(* Logix 5000 project; controller RSL5k_18_Template_noLib Emulate 5570 rev 32.11; software revision 32.02; part 3 of 16 *)
(* tags used below, declared in another part *)
   PCmd_ClearCapt : BOOL;   // Program Command to Clear the captured min / max PV excursion values
   P_AIn : BOOL;   // Unique Parameter Name for auto - discovery
   Wrk_ValidONS : BOOL;   // Selected PV goes from Infinite or Not a Number to VALID
   OCmd_ResetAckAll : BOOL;   // Operator Command to Reset and Acknowledge all Alarms
   MCmd_InpPV : BOOL;   // Maintenance Command to use Input PV (normal)
   MCmd_SubstPV : BOOL;   // Maintenance Command to use Substitute PV (override input)
(* P_AIn, continued *)

ROUTINE Prescan   (* ladder *)
// Clear Ownership. clear "lurking" Commands
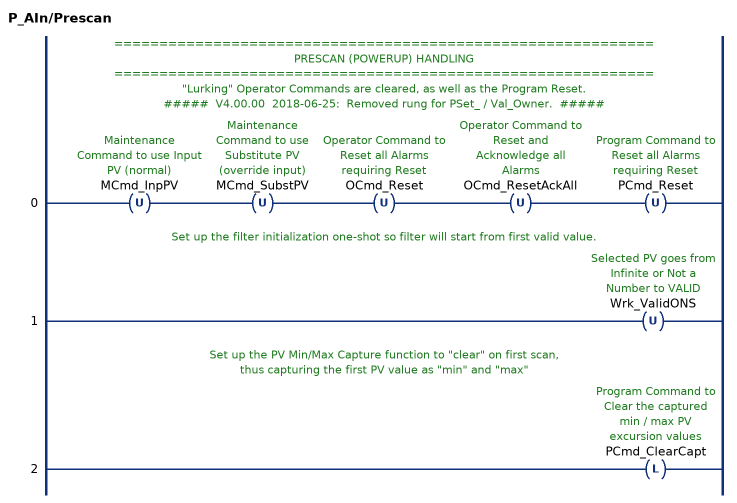
   // ============================================================
   // PRESCAN (POWERUP) HANDLING
   // ============================================================
   // "Lurking" Operator Commands are cleared, as well as the Program Reset.
   // #####  V4.00.00  2018-06-25:  Removed rung for PSet_ / Val_Owner.  #####
   0: OTU(MCmd_InpPV)OTU(MCmd_SubstPV)OTU(OCmd_Reset)OTU(OCmd_ResetAckAll)OTU(PCmd_Reset);
   // Set up the filter initialization one-shot so filter will start from first valid value.
   1: OTU(Wrk_ValidONS);
   // Set up the PV Min/Max Capture function to "clear" on first scan,
   // thus capturing the first PV value as "min" and "max"
   2: OTL(PCmd_ClearCapt);
END_ROUTINE
END_ADD_ON_INSTRUCTION

ADD_ON_INSTRUCTION P_Alarm   (* revision 4.10 .00 Release, vendor Rockwell Automation, ExecutePrescan, ExecuteEnableInFalse *)
// Alarm
// Revision note:
// See Instruction Help for a summary of changes, and see 4.10 Release Notes for details.
// Help:
// Copyright © Rockwell Automation, Inc.  All Rights Reserved.
// This instruction monitors one input condition and provides one Alarm with:
//   * configurable latching (reset required) and acknowledgement requirement
//   * configurable alarm severity
//       1 to 250       = Low  (blue, typ. informational)
//       251 to 500   = Medium  (yelllow, typ. warning)
//       501 to 750   = High  (red, typ. process exception)
//       751 to 1000 = Urgent  (magenta, typ. equip. fault)
//   * configurable minimum ON time (e.g., to ensure it is seen by the HMI)
//   * commands to suppress/unsuppress (Prog), shelve/unshelve (Oper)
//         and disable/enable (Maint) the alarm.
//   * configurable amount of time shelved to automatically unshelve an alarm
//   * FTA&E support for suppressed, shelved and disabled states (V7.0)
//   * a Maintenance "Test" command, which triggers the alarm for the minimum
//      alarm time for testing purposes.
// NOTE regarding parameter naming:
//   FTAE names (same as ALMD instruction) are used instead
//   of the ANSI/ISA 18.2-2009 names, as follows:
//    "Disabled" is the equivalent of "Out of Service" in ISA 18.2.
//       (The Disabled state is owned by Maintenance.)
//    "Suppressed" is the equivalent of "Suppressed by Design" in
//       ISA 18.2. (The Suppressed state is owned by Program logic.)
//    "Shelved" is the same as in ISA 18.2.
//       (The Shelved state is owned by Operator, but may be cleared
//       by Program logic based on time, shift change, etc.)
// This instruction is usually nested within other instructions, with one instance
// used for each Alarm generated by the containing instruction.  It may also be
// used as a standalone instruction for Alarm conditions generated by custom logic.
// FTAE Alarm Setup:
//   (object).(alarm).Com_AE.0:  Alarm to FTAE
//     .Com_AE.1:   Ack to/from FTAE
//     .Com_AE.3:   Shelved from FTAE Status
//     .Com_AE.4:   Shelve/Reshelve to FTAE Control (auto reset)
//     .Com_AE.5:   Unshelve to FTAE Control (auto reset)
//     .Com_AE.6:   Suppressed from FTAE Status
//     .Com_AE.7:   Suppress to FTAE Control (auto reset)
//     .Com_AE.8:   Unsuppress to FTAE Control (auto reset)
//     .Com_AE.9:   Disabled from FTAE Status
//     .Com_AE.10: Disable to FTAE Control (auto reset)
//     .Com_AE.11: Enable to FTAE Control (auto reset)
//    all other bits unused
//     .Cfg_MaxShelfT is also used in FTAE config.
//     .Cfg_Severity is used in FTAE for FTView 8.x and later.
// SUMMARY OF CHANGES FROM PREVIOUS VERSION (4.00.00)
// See 4.10 Release Notes for details.
// * Unmodified, up-rev only for Library 4.10.00
// SUMMARY OF CHANGES FROM PREVIOUS VERSION (3.5-07 Patch01)
// See 4.00 Release Notes for details.
// * Changed Inf_Lib and Inf_Type to HMI_Lib and HMI_Type.
// * Deleted Cfg_PCmdClear.  All Program Commands are now self-clearing.
// * Aligned ready bit naming with command bit names.
// * All OCmds/MCmds and ORdys/MRdys are now Local Tags.
// * Added Sts_RdyAck and Sts_RdyReset for use by containing objects.
// * Modified to remove Suppressed from the conditions which show the
//     "Inhibited" breadcrumb.
// * Added Inp_OoS for Out of Service from parent object's P_CmdSrc.
VAR_INPUT
   Inp : BOOL := 1; {visible}   // Alarm Condition Input 1=Alarm
   Inp_OoS : ALIAS FOR Com_AE.2;   // 1=Out of Service (from object's P_CmdSrc)
   Inp_Reset : BOOL; {visible}   // 1=Reset Alarm requiring reset
   Cfg_Exists : BOOL := 1;   // 1=Alarm configured to exist, 0=Does not exist, don't scan
   Cfg_ResetReqd : BOOL;   // 1=Latched Alarm, a Reset is required to clear this Alarm
   Cfg_AckReqd : BOOL := 1;   // 1=Acknowledge required for this Alarm
   Cfg_AllowShelve : BOOL := 1;   // 1=Allow Operator to Shelve this Alarm
   Cfg_AllowDisable : BOOL := 1;   // 1=Allow Maintenance to Disable this Alarm
   Cfg_Severity : DINT := 750;   // Alarm Severity: 1..250=Low, 251..500=Medium, 501..750=High, 751..1000=Urgent
   Cfg_MaxShelfT : DINT := 480;   // Auto unshelve after shelved this long (1..32767 minutes)
   Cfg_AlmMinOnT : DINT := 5;   // Minimum time Alm output stays on (sec)
   PCfg_AllowExist : BOOL := 1;   // 1=Alarm can be configured to exist, 0=other configs make alarm meaningless
   PCmd_Reset : BOOL;   // Program Command to Reset latched alarm
   PCmd_Ack : BOOL;   // Program Command to Acknowledge alarm
   PCmd_Suppress : BOOL;   // Program Command to Suppress by Design (inhibits new alarm)
   PCmd_Unsuppress : BOOL;   // Program Command to Unsuppress (allows new alarm)
   PCmd_Unshelve : BOOL;   // Program Command to Unshelve (e.g., on shift change)
END_VAR
VAR_OUTPUT
   Val_Notify : DINT; {access Read Only}   // Current Alarm Severity and Acknowledgement (enumeration)
   Val_SecToUnshelve : DINT; {access Read Only, visible}   // Number of Seconds until this alarm unshelves itself (mmm:ss)
   Val_MinToUnshelve : DINT; {access Read Only, visible}   // Number of minutes until this alarm unshelves itself (mmm:ss)
   Alm : ALIAS FOR Com_AE.0; {visible}   // Alarm output 1=In Alarm
   Ack : ALIAS FOR Com_AE.1; {visible}   // Alarm acknowledged status: 1=Ack rcvd
   Shelved : ALIAS FOR Com_AE.3; {visible}   // 1=Alarm has been Shelved by Operator (inhibits new alarm)
   Suppressed : ALIAS FOR Com_AE.6; {visible}   // 1=Alarm has been Suppressed by Program (inhibits new alarm)
   Disabled : ALIAS FOR Com_AE.9; {visible}   // 1=Alarm has been Disabled by Maintanance (inhibits new alarm)
   Sts_AlmInh : BOOL; {access Read Only}   // 1=Alarm has been suppressed, shelved or disabled, display "I" icon
   Sts_RdyReset : ALIAS FOR ORdy_Reset; {access Read Only}   // 1=A latched alarm or shed condition is ready to be reset
   Sts_RdyAck : ALIAS FOR ORdy_Ack; {access Read Only}   // 1=An alarm is ready to be acknowledged
   Sts_Err : BOOL; {access Read Only}   // 1=Error in Config: see detail Err_ bits for reason
   Err_Timer : BOOL; {access Read Only}   // 1=Error in Config: Alarm Min On Time, Shelf Time (use 0 to 2147483)
   Err_Severity : BOOL; {access Read Only}   // 1=Error in Config: Invalid Severity (use 1 to 4)
   P_Alarm : BOOL;   // Unique Parameter Name for auto - discovery
END_VAR
VAR
   Wrk_Alm : BOOL; {access None}   // Internal Alarm Status
   Wrk_Suppressed : BOOL; {access None}   // Internal Alarm Suppressed Status
   Wrk_AlmMinOnT : TIMER := (PRE := 5000); {access None}   // Alarm output minimum ON time to be seen by alarm server
   Wrk_AutoAckT : TIMER := (PRE := 5000); {access None}   // Time to clear Ack bit when Ack not required
   Wrk_ShelfT : TIMER; {access Read Only}   // Time to auto Unshelve a Shelved Alarm
   HMI_Tab : SINT;   // Tab to display (FTView ME)
   Com_AE : INT := 2#0000_0000_0000_0010;   // Communication with HMI / Alarm/Event Server (see bit descriptions)
        .0   // Alarm to AE
        .10   // Disable to AE Control
        .11   // Enable to AE Control
        .12   // (not used)
        .13   // (not used)
        .14   // (not used)
        .15   // (not used)
        .1   // Acked from AE Status, Ack to AE Control
        .2   // Out of Service (from parent object's P_CmdSrc)
        .3   // Shelved from AE Status
        .4   // Shelve to AE Control
        .5   // Unshelve to AE Control
        .6   // Suppressed from AE Status
        .7   // Suppress to AE Control
        .8   // Unsuppress to AE Control
        .9   // Disabled from AE Status
   Cfg_Tag : STRING_20 := 'P_Alarm';   // Alarm Tag Text (e.g., "LAHH-101")
   Cfg_Cond : STRING_20 := 'Alarm Condition';   // Alarm Condition Text (e.g., "High-High PV")
   Wrk_SecToUnshelve : DINT; {access None}   // Number of seconds until this alarm unshelves itself
   HMI_Lib : STRING_12 := 'RA-BAS'; {access Read Only}   // Display Library for Faceplate call-up
   HMI_Type : STRING_16 := 'P_Alarm'; {access Read Only}   // Must contain AOI name, used for HMI and Information S/W
   ORdy_Unshelve : BOOL; {access Read Only}   // 1=Ready for OCmd_Unshelve (enables HMI button)
   ORdy_Shelve : BOOL; {access Read Only}   // 1=Ready for OCmd_Shelve (enables HMI button)
   MRdy_Test : BOOL; {access Read Only}   // 1=Ready for MCmd_Test (enables HMI button)
   MRdy_Enable : BOOL; {access Read Only}   // 1=Ready for MCmd_Enable (enables HMI button)
   MRdy_Disable : BOOL; {access Read Only}   // 1=Ready for MCmd_Disable (enables HMI button)
   OCmd_Unshelve : BOOL;   // Operator Command to Unshelve alarm (allows new alarm)
   OCmd_Shelve : BOOL;   // Operator Command to Shelve Alarm (inhibits new alarm)
   OCmd_Ack : BOOL;   // Operator Command to Acknowledge alarm
   OCmd_Reset : BOOL;   // Operator Command to Reset latched alarm
   MCmd_Test : BOOL;   // Maintenance Command to Test alarm (issued for minimum alarm time)
   MCmd_Enable : BOOL;   // Maintenance Command to Enable alarm (allows new alarm)
   MCmd_Disable : BOOL;   // Maintenance Command to Disable alarm (inhibits new alarm)
   ORdy_Ack : BOOL; {access Read Only}   // 1=Ready for OCmd_Ack (enables HMI button)
   ORdy_Reset : BOOL; {access Read Only}   // 1=Ready for OCmd_Reset (enables HMI button)
END_VAR

ROUTINE EnableInFalse   (* ladder *)
// Perform Alarm processing, but Invert Alarm Input ("Inp") for use on LD rung (EnableIn False)
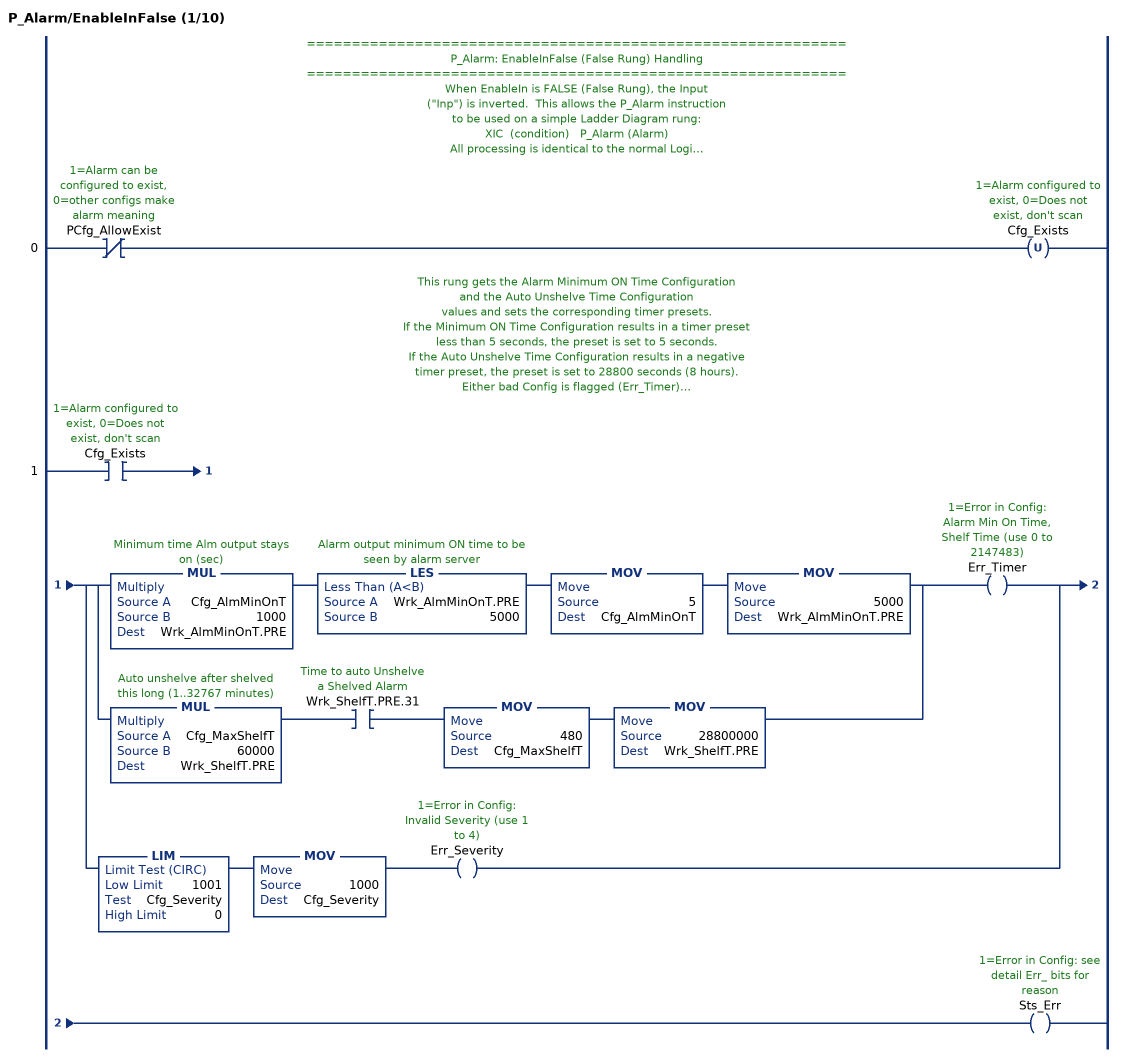
   // ============================================================
   // P_Alarm: EnableInFalse (False Rung) Handling
   // ============================================================
   // When EnableIn is FALSE (False Rung), the Input
   // ("Inp") is inverted.  This allows the P_Alarm instruction
   // to be used on a simple Ladder Diagram rung:
   // XIC  (condition)   P_Alarm (Alarm)
   // All processing is identical to the normal Logic
   // routine, except references to Inp are inverted!
   // ============================================================
   // CONFIGURATION
   // ============================================================
   // In the object containing this alarm, other configuration (such as not having
   // any limit switches) may make this particular alarm meaningless.
   // The Program Configuration "Allow Exist" is used to hide this alarm
   // on the object's faceplate and other graphics, and forces the Cfg_Exist to 0.
   0: XIO(PCfg_AllowExist)OTU(Cfg_Exists);
   // This rung gets the Alarm Minimum ON Time Configuration
   // and the Auto Unshelve Time Configuration
   // values and sets the corresponding timer presets.
   // If the Minimum ON Time Configuration results in a timer preset
   // less than 5 seconds, the preset is set to 5 seconds.
   // If the Auto Unshelve Time Configuration results in a negative
   // timer preset, the preset is set to 28800 seconds (8 hours).
   // Either bad Config is flagged (Err_Timer).
   // Bad Config is also flagged if the Cfg_Severity is out of range (valid = 1..1000) (Err_Severity).
   1: XIC(Cfg_Exists)[[MUL(Cfg_AlmMinOnT,1000,Wrk_AlmMinOnT.PRE) LES(Wrk_AlmMinOnT.PRE,5000) MOV(5,Cfg_AlmMinOnT) MOV(5000,Wrk_AlmMinOnT.PRE) ,MUL(Cfg_MaxShelfT,60000,Wrk_ShelfT.PRE) XIC(Wrk_ShelfT.PRE.31) MOV(480,Cfg_MaxShelfT) MOV(28800000,Wrk_ShelfT.PRE) ] OTE(Err_Timer) ,LIM(1001,Cfg_Severity,0) MOV(1000,Cfg_Severity) OTE(Err_Severity) ]OTE(Sts_Err);
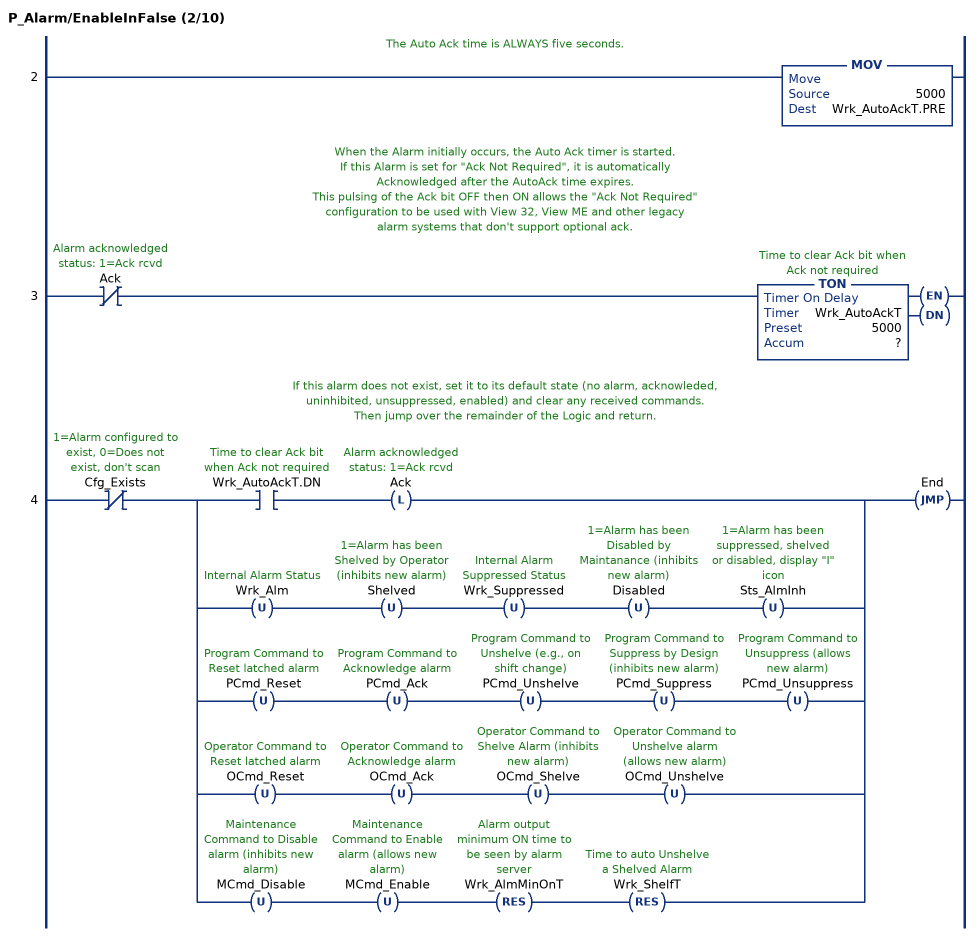
   // The Auto Ack time is ALWAYS five seconds.
   2: MOV(5000,Wrk_AutoAckT.PRE);
   // When the Alarm initially occurs, the Auto Ack timer is started.
   // If this Alarm is set for "Ack Not Required", it is automatically
   // Acknowledged after the AutoAck time expires.
   // This pulsing of the Ack bit OFF then ON allows the "Ack Not Required"
   // configuration to be used with View 32, View ME and other legacy
   // alarm systems that don't support optional ack.
   3: XIO(Ack)TON(Wrk_AutoAckT,?,?);
   // If this alarm does not exist, set it to its default state (no alarm, acknowleded,
   // uninhibited, unsuppressed, enabled) and clear any received commands.
   // Then jump over the remainder of the Logic and return.
   4: XIO(Cfg_Exists)[XIC(Wrk_AutoAckT.DN) OTL(Ack) ,OTU(Wrk_Alm) OTU(Shelved) OTU(Wrk_Suppressed) OTU(Disabled) OTU(Sts_AlmInh) ,OTU(PCmd_Reset) OTU(PCmd_Ack) OTU(PCmd_Unshelve) OTU(PCmd_Suppress) OTU(PCmd_Unsuppress) ,OTU(OCmd_Reset) OTU(OCmd_Ack) OTU(OCmd_Shelve) OTU(OCmd_Unshelve) ,OTU(MCmd_Disable) OTU(MCmd_Enable) RES(Wrk_AlmMinOnT) RES(Wrk_ShelfT) ]JMP(End);
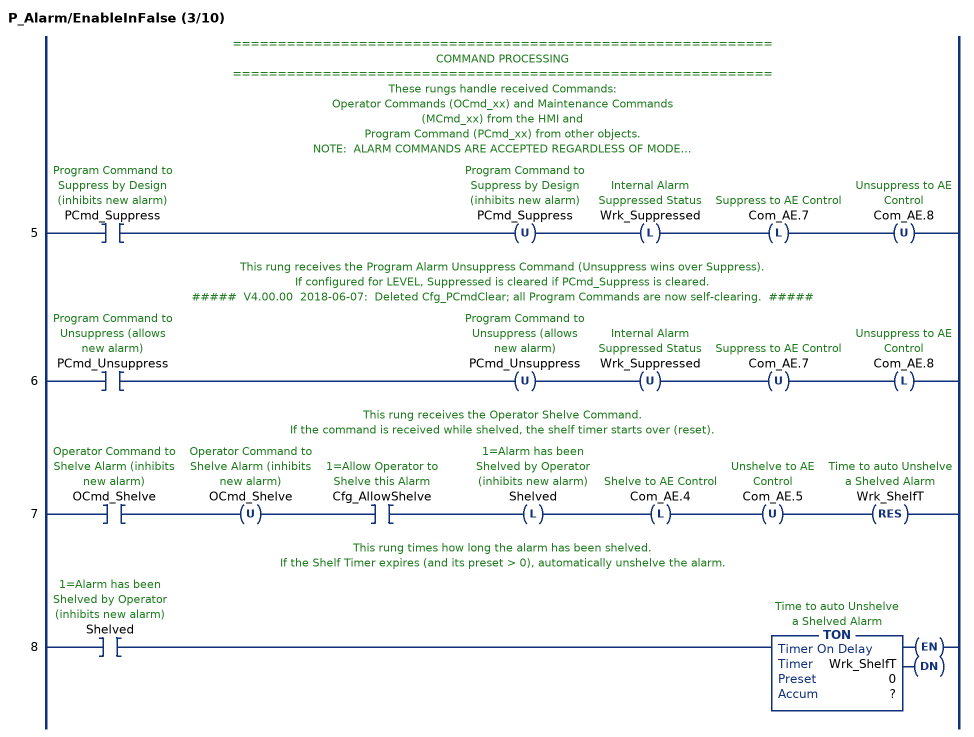
   // ============================================================
   // COMMAND PROCESSING
   // ============================================================
   // These rungs handle received Commands:
   // Operator Commands (OCmd_xx) and Maintenance Commands
   // (MCmd_xx) from the HMI and
   // Program Command (PCmd_xx) from other objects.
   // NOTE:  ALARM COMMANDS ARE ACCEPTED REGARDLESS OF MODE.
   // This rung receives the Program Alarm Inhibit Command.
   // If configured for EDGE, the Command is cleared.
   // #####  V4.00.00  2018-06-07:  Deleted Cfg_PCmdClear; all Program Commands are now self-clearing.  #####
   5: XIC(PCmd_Suppress)OTU(PCmd_Suppress)OTL(Wrk_Suppressed)OTL(Com_AE.7)OTU(Com_AE.8);
   // This rung receives the Program Alarm Unsuppress Command (Unsuppress wins over Suppress).
   // If configured for LEVEL, Suppressed is cleared if PCmd_Suppress is cleared.
   // #####  V4.00.00  2018-06-07:  Deleted Cfg_PCmdClear; all Program Commands are now self-clearing.  #####
   6: XIC(PCmd_Unsuppress)OTU(PCmd_Unsuppress)OTU(Wrk_Suppressed)OTU(Com_AE.7)OTL(Com_AE.8);
   // This rung receives the Operator Shelve Command.
   // If the command is received while shelved, the shelf timer starts over (reset).
   7: XIC(OCmd_Shelve)OTU(OCmd_Shelve)XIC(Cfg_AllowShelve)OTL(Shelved)OTL(Com_AE.4)OTU(Com_AE.5)RES(Wrk_ShelfT);
   // This rung times how long the alarm has been shelved.
   // If the Shelf Timer expires (and its preset > 0), automatically unshelve the alarm.
   8: XIC(Shelved)TON(Wrk_ShelfT,?,?);
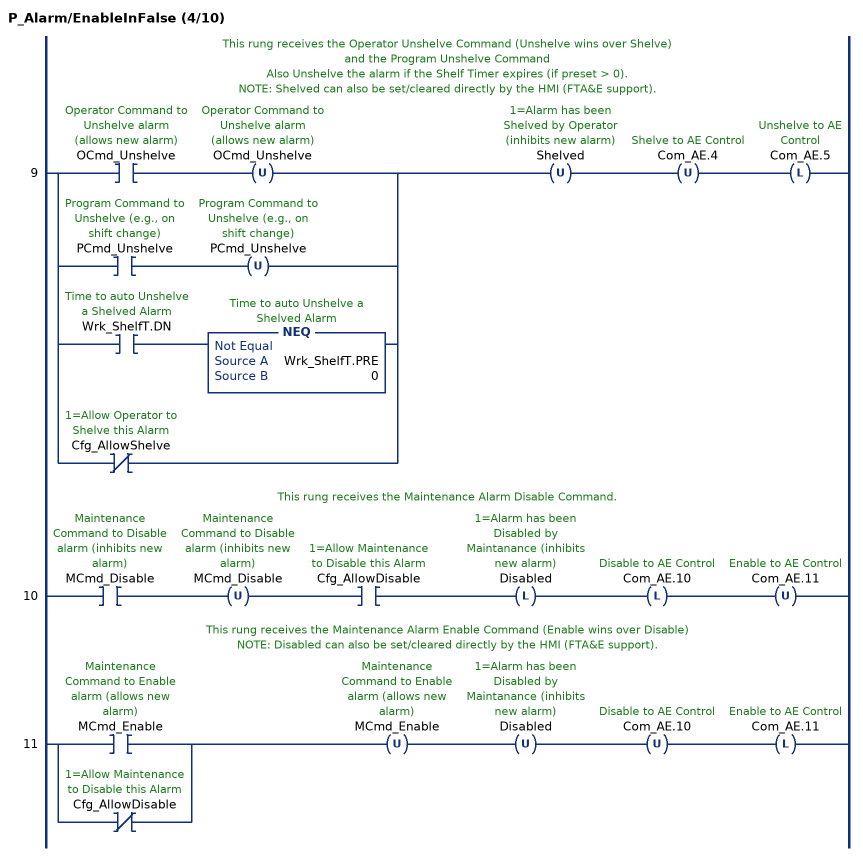
   // This rung receives the Operator Unshelve Command (Unshelve wins over Shelve)
   // and the Program Unshelve Command
   // Also Unshelve the alarm if the Shelf Timer expires (if preset > 0).
   // NOTE: Shelved can also be set/cleared directly by the HMI (FTA&E support).
   9: [XIC(OCmd_Unshelve) OTU(OCmd_Unshelve) ,XIC(PCmd_Unshelve) OTU(PCmd_Unshelve) ,XIC(Wrk_ShelfT.DN) NEQ(Wrk_ShelfT.PRE,0) ,XIO(Cfg_AllowShelve) ]OTU(Shelved)OTU(Com_AE.4)OTL(Com_AE.5);
   // This rung receives the Maintenance Alarm Disable Command.
   10: XIC(MCmd_Disable)OTU(MCmd_Disable)XIC(Cfg_AllowDisable)OTL(Disabled)OTL(Com_AE.10)OTU(Com_AE.11);
   // This rung receives the Maintenance Alarm Enable Command (Enable wins over Disable)
   // NOTE: Disabled can also be set/cleared directly by the HMI (FTA&E support).
   11: [XIC(MCmd_Enable) ,XIO(Cfg_AllowDisable) ]OTU(MCmd_Enable)OTU(Disabled)OTU(Com_AE.10)OTL(Com_AE.11);
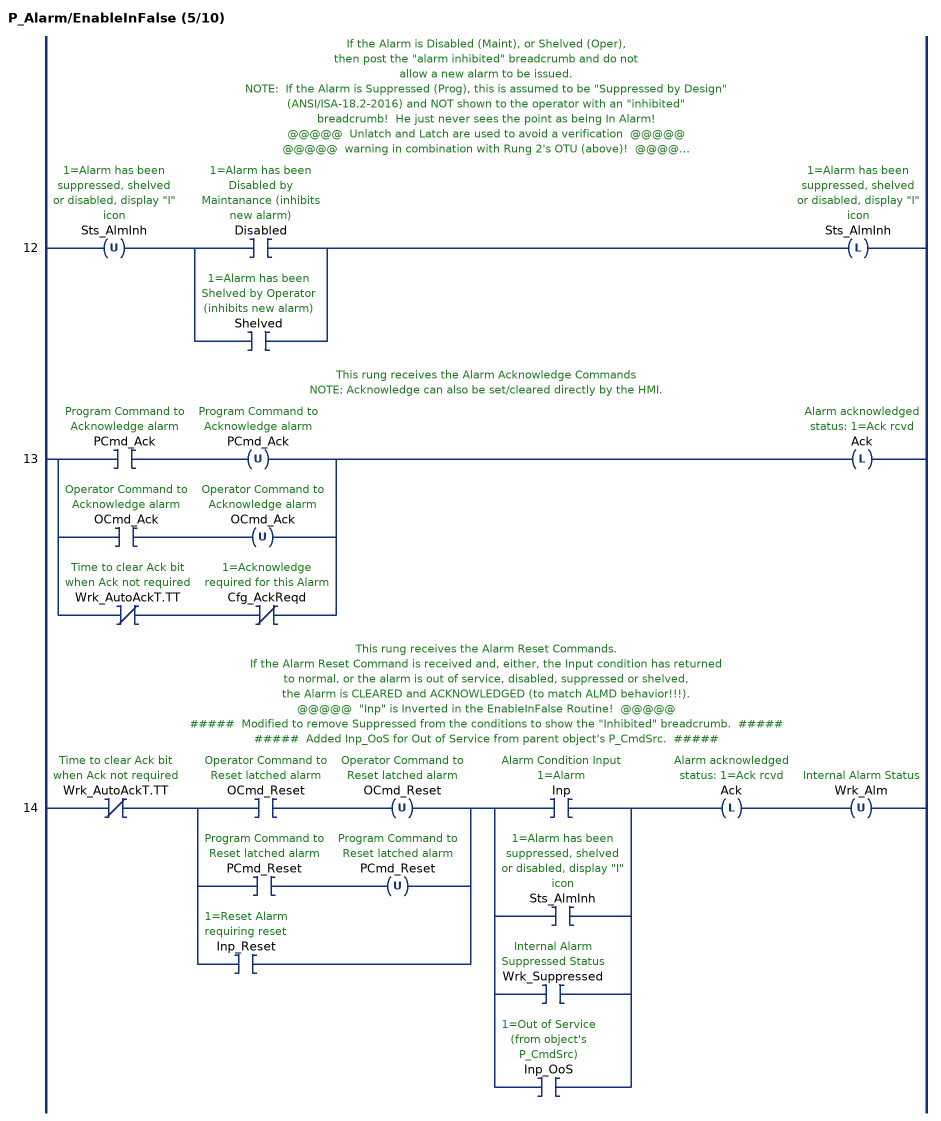
   // If the Alarm is Disabled (Maint), or Shelved (Oper),
   // then post the "alarm inhibited" breadcrumb and do not
   // allow a new alarm to be issued.
   // NOTE:  If the Alarm is Suppressed (Prog), this is assumed to be "Suppressed by Design"
   // (ANSI/ISA-18.2-2016) and NOT shown to the operator with an "inhibited"
   // breadcrumb!  He just never sees the point as being In Alarm!
   // @@@@@  Unlatch and Latch are used to avoid a verification  @@@@@
   // @@@@@  warning in combination with Rung 2's OTU (above)!  @@@@@
   // #####  V4.00.00  2018-06-07:  Modified to remove Suppressed from the conditions to show the "Inhibited" breadcrumb.  #####
   12: OTU(Sts_AlmInh)[XIC(Disabled) ,XIC(Shelved) ]OTL(Sts_AlmInh);
   // This rung receives the Alarm Acknowledge Commands
   // NOTE: Acknowledge can also be set/cleared directly by the HMI.
   13: [XIC(PCmd_Ack) OTU(PCmd_Ack) ,XIC(OCmd_Ack) OTU(OCmd_Ack) ,XIO(Wrk_AutoAckT.TT) XIO(Cfg_AckReqd) ]OTL(Ack);
   // This rung receives the Alarm Reset Commands.
   // If the Alarm Reset Command is received and, either, the Input condition has returned
   // to normal, or the alarm is out of service, disabled, suppressed or shelved,
   // the Alarm is CLEARED and ACKNOWLEDGED (to match ALMD behavior!!!).
   // @@@@@  "Inp" is Inverted in the EnableInFalse Routine!  @@@@@
   // #####  Modified to remove Suppressed from the conditions to show the "Inhibited" breadcrumb.  #####
   // #####  Added Inp_OoS for Out of Service from parent object's P_CmdSrc.  #####
   14: XIO(Wrk_AutoAckT.TT)[XIC(OCmd_Reset) OTU(OCmd_Reset) ,XIC(PCmd_Reset) OTU(PCmd_Reset) ,XIC(Inp_Reset) ][XIC(Inp) ,XIC(Sts_AlmInh) ,XIC(Wrk_Suppressed) ,XIC(Inp_OoS) ]OTL(Ack)OTU(Wrk_Alm);
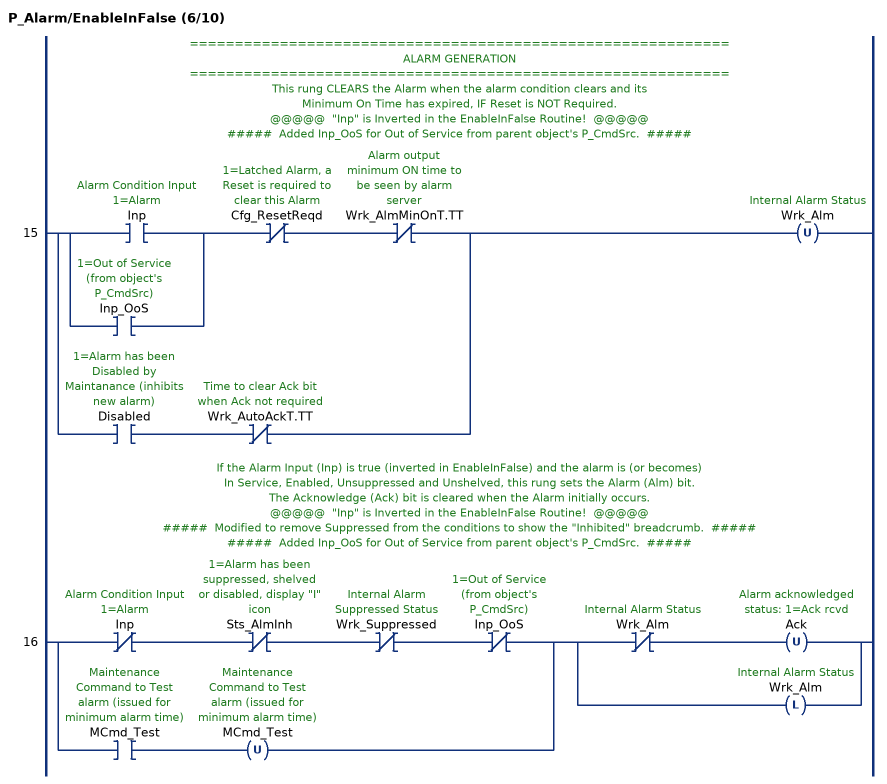
   // ============================================================
   // ALARM GENERATION
   // ============================================================
   // This rung CLEARS the Alarm when the alarm condition clears and its
   // Minimum On Time has expired, IF Reset is NOT Required.
   // @@@@@  "Inp" is Inverted in the EnableInFalse Routine!  @@@@@
   // #####  Added Inp_OoS for Out of Service from parent object's P_CmdSrc.  #####
   15: [[XIC(Inp) ,XIC(Inp_OoS) ] XIO(Cfg_ResetReqd) XIO(Wrk_AlmMinOnT.TT) ,XIC(Disabled) XIO(Wrk_AutoAckT.TT) ]OTU(Wrk_Alm);
   // If the Alarm Input (Inp) is true (inverted in EnableInFalse) and the alarm is (or becomes)
   // In Service, Enabled, Unsuppressed and Unshelved, this rung sets the Alarm (Alm) bit.
   // The Acknowledge (Ack) bit is cleared when the Alarm initially occurs.
   // @@@@@  "Inp" is Inverted in the EnableInFalse Routine!  @@@@@
   // #####  Modified to remove Suppressed from the conditions to show the "Inhibited" breadcrumb.  #####
   // #####  Added Inp_OoS for Out of Service from parent object's P_CmdSrc.  #####
   16: [XIO(Inp) XIO(Sts_AlmInh) XIO(Wrk_Suppressed) XIO(Inp_OoS) ,XIC(MCmd_Test) OTU(MCmd_Test) ][XIO(Wrk_Alm) OTU(Ack) ,OTL(Wrk_Alm) ];
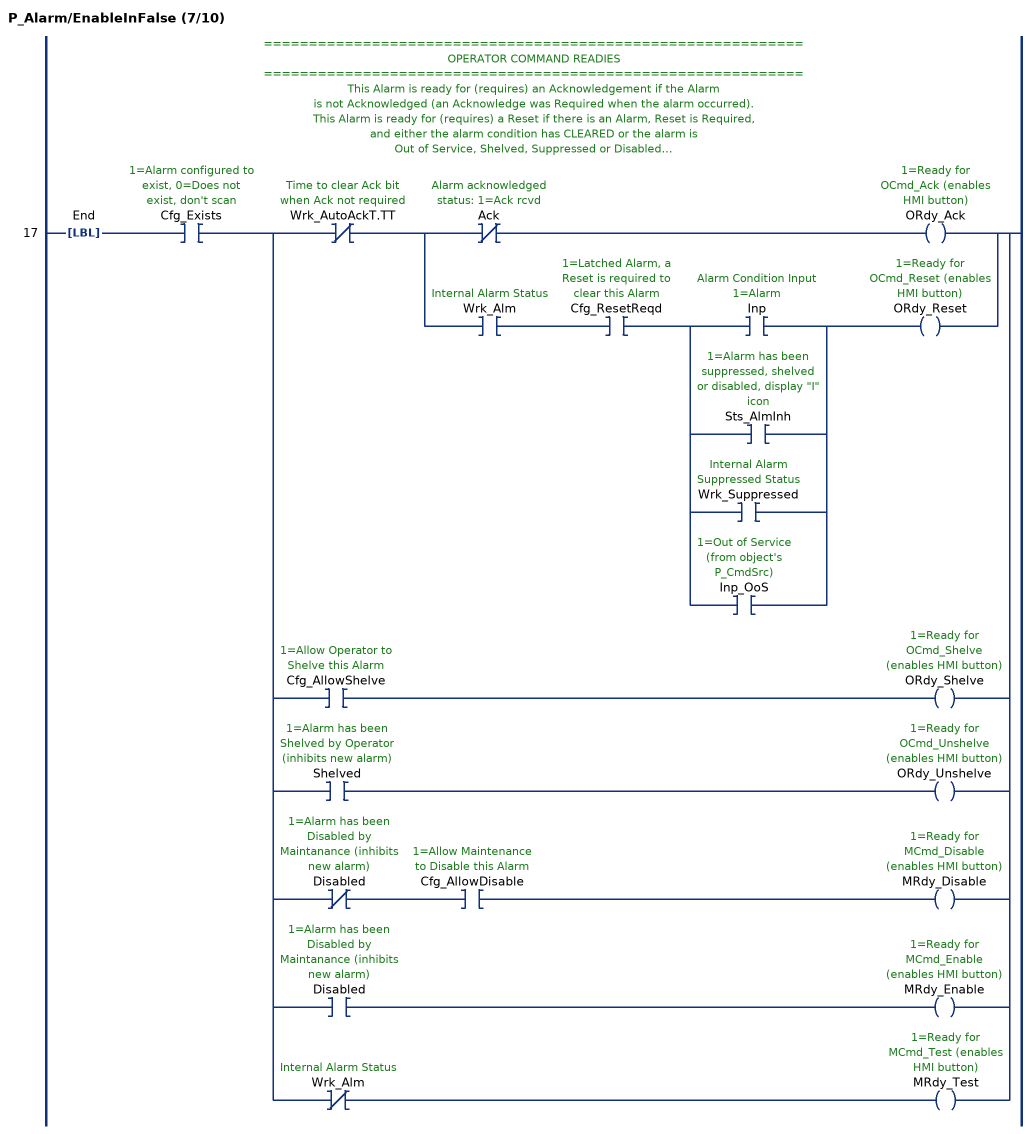
   // ============================================================
   // OPERATOR COMMAND READIES
   // ============================================================
   // This Alarm is ready for (requires) an Acknowledgement if the Alarm
   // is not Acknowledged (an Acknowledge was Required when the alarm occurred).
   // This Alarm is ready for (requires) a Reset if there is an Alarm, Reset is Required,
   // and either the alarm condition has CLEARED or the alarm is
   // Out of Service, Shelved, Suppressed or Disabled.
   // .
   // If the Alarm is NOT Shelved, it is ready for Shelve.
   // If the Alarm IS Shelved, it is ready for Unshelve.
   // If the Alarm is NOT Disabled, it is ready for Disable.
   // If the Alarm IS Disabled, it is ready for Enable.
   // NOTE: This rung appears before the Values/Status rung because the Rdy_Reset
   // condition is used to eliminate redundant logic in the rung below for Val_Notify.0.
   // @@@@@  "Inp" is Inverted in the EnableInFalse Routine!  @@@@@
   // #####  V4.00.00  2018-06-07:  Aligned ready bit naming with command bit names.  #####
   // #####  All OCmds/MCmds and ORdys/MRdys are now Local Tags.  #####
   // #####  Added Sts_RdyAck and Sts_ResetReqd for use by containing objects.  #####
   // #####  Modified to remove Suppressed from the conditions to show the "Inhibited" breadcrumb.  #####
   // #####  Added Inp_OoS for Out of Service from parent object's P_CmdSrc.  #####
   17: LBL(End)XIC(Cfg_Exists)[XIO(Wrk_AutoAckT.TT) [XIO(Ack) OTE(ORdy_Ack) ,XIC(Wrk_Alm) XIC(Cfg_ResetReqd) [XIC(Inp) ,XIC(Sts_AlmInh) ,XIC(Wrk_Suppressed) ,XIC(Inp_OoS) ] OTE(ORdy_Reset) ] ,XIC(Cfg_AllowShelve) OTE(ORdy_Shelve) ,XIC(Shelved) OTE(ORdy_Unshelve) ,XIO(Disabled) XIC(Cfg_AllowDisable) OTE(MRdy_Disable) ,XIC(Disabled) OTE(MRdy_Enable) ,XIO(Wrk_Alm) OTE(MRdy_Test) ];
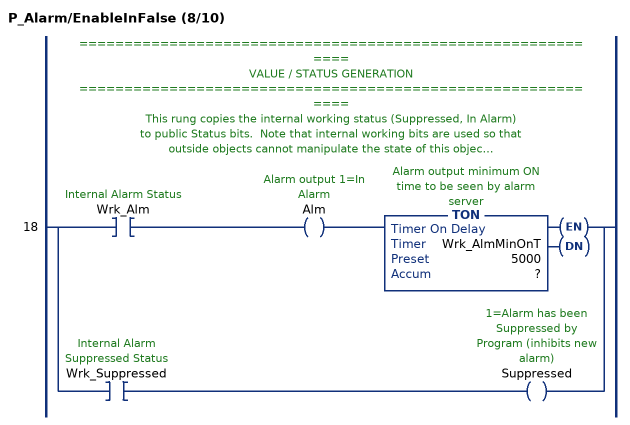
   // ============================================================
   // VALUE / STATUS GENERATION
   // ============================================================
   // This rung copies the internal working status (Suppressed, In Alarm)
   // to public Status bits.  Note that internal working bits are used so that
   // outside objects cannot manipulate the state of this object
   // by setting/clearing its Status and Alarm bits.
   // Public Status is generated for:
   // Alarm (with minimum ON time to be seen by polling)
   // Alarm Suppressed
   // Unsuppressed, Unshelved and Enabled are generated for HMI (FTVSE 7).
   // (Ack, Shelved and Disabled can be set/cleared by the HMI directly.
   // Note that these bits are "read/write" outputs in the parameter definition.)
   18: [XIC(Wrk_Alm) OTE(Alm) TON(Wrk_AlmMinOnT,?,?) ,XIC(Wrk_Suppressed) OTE(Suppressed) ];
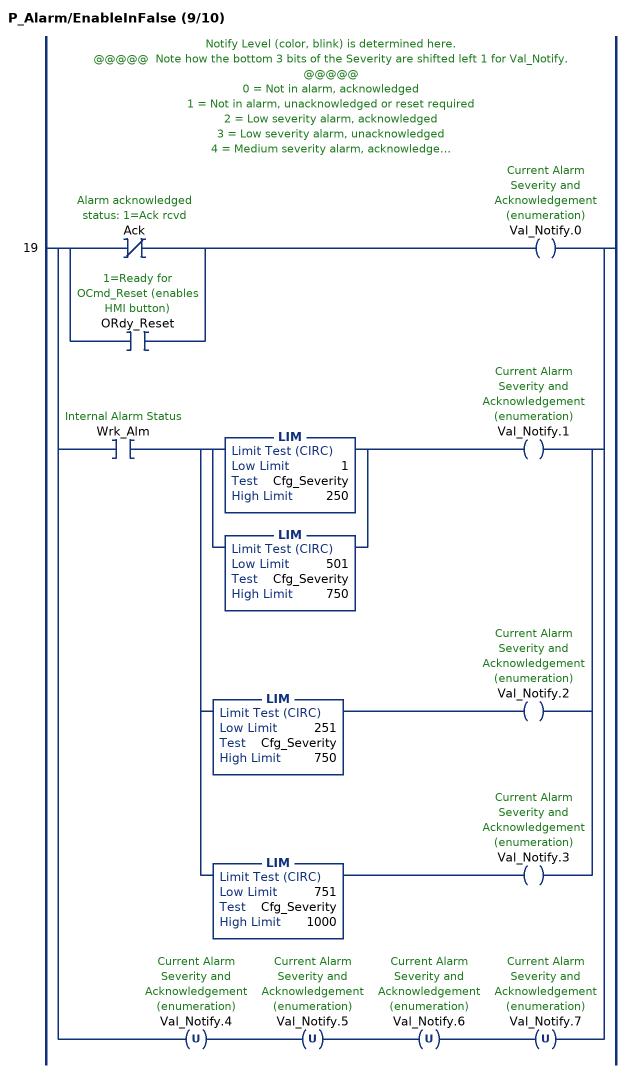
   // Notify Level (color, blink) is determined here.
   // @@@@@  Note how the bottom 3 bits of the Severity are shifted left 1 for Val_Notify.  @@@@@
   // 0 = Not in alarm, acknowledged
   // 1 = Not in alarm, unacknowledged or reset required
   // 2 = Low severity alarm, acknowledged
   // 3 = Low severity alarm, unacknowledged
   // 4 = Medium severity alarm, acknowledged
   // 5 = Medium severity alarm, unacknowledged
   // 6 = High severity alarm, acknowledged
   // 7 = High severity alarm, unacknowledged
   // 8 = Urgent severity alarm, acknowledged
   // 9 = Urgent severity alarm, unacknowledged
   // NOTE that the alarm bell icon will blink, even though the alarm is Acknowledged,
   // if an Alarm Reset is required (to get the Operator's attention).
   19: [[XIO(Ack) ,XIC(ORdy_Reset) ] OTE(Val_Notify.0) ,XIC(Wrk_Alm) [[LIM(1,Cfg_Severity,250) ,LIM(501,Cfg_Severity,750) ] OTE(Val_Notify.1) ,LIM(251,Cfg_Severity,750) OTE(Val_Notify.2) ,LIM(751,Cfg_Severity,1000) OTE(Val_Notify.3) ] ,OTU(Val_Notify.4) OTU(Val_Notify.5) OTU(Val_Notify.6) OTU(Val_Notify.7) ];
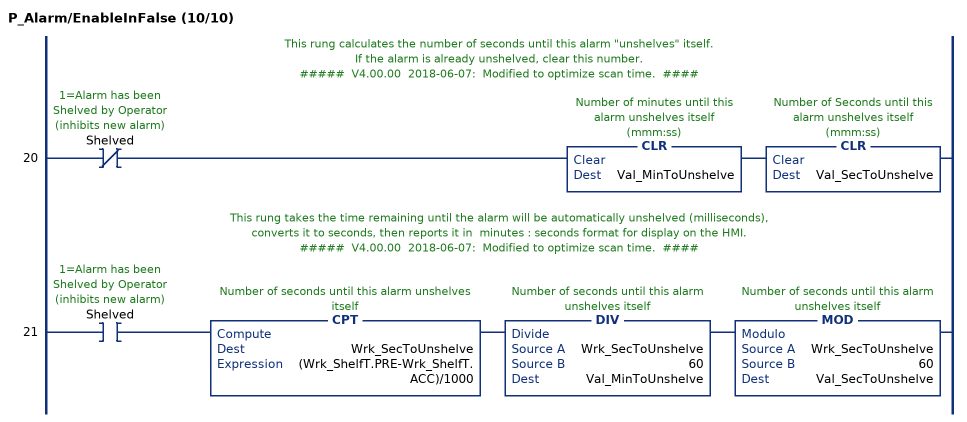
   // This rung calculates the number of seconds until this alarm "unshelves" itself.
   // If the alarm is already unshelved, clear this number.
   // #####  V4.00.00  2018-06-07:  Modified to optimize scan time.  ####
   20: XIO(Shelved)CLR(Val_MinToUnshelve)CLR(Val_SecToUnshelve);
   // This rung takes the time remaining until the alarm will be automatically unshelved (milliseconds),
   // converts it to seconds, then reports it in  minutes : seconds format for display on the HMI.
   // #####  V4.00.00  2018-06-07:  Modified to optimize scan time.  ####
   21: XIC(Shelved)CPT(Wrk_SecToUnshelve,(Wrk_ShelfT.PRE-Wrk_ShelfT.ACC)/1000)DIV(Wrk_SecToUnshelve,60,Val_MinToUnshelve)MOD(Wrk_SecToUnshelve,60,Val_SecToUnshelve);
END_ROUTINE

ROUTINE Logic   (* ladder *)
// Perform Alarm processing: delay, latch/reset, acknowledge, enable/disable, inhibit/uninhibit, suppress/unsuppress
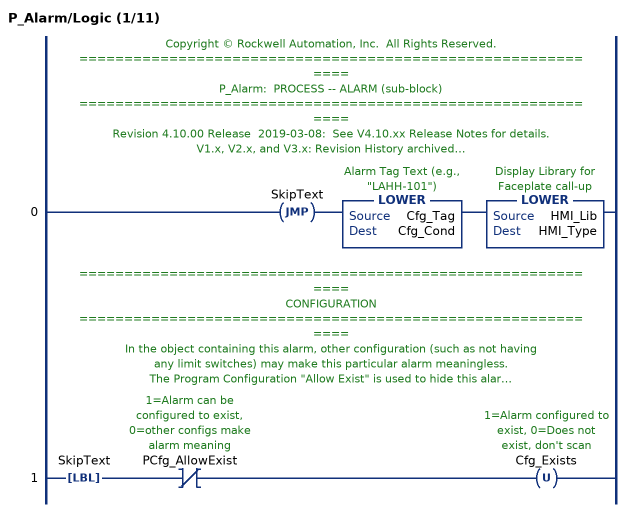
   // Copyright © Rockwell Automation, Inc.  All Rights Reserved.
   // ============================================================
   // P_Alarm:  PROCESS -- ALARM (sub-block)
   // ============================================================
   // Revision 4.10.00 Release  2019-03-08:  See V4.10.xx Release Notes for details.
   // V1.x, V2.x, and V3.x: Revision History archived.
   // V4.00.00  2018-06-07:  Changed Inf_ items to HMI_. Deleted Cfg_PCmdClear.
   // Aligned ready bit naming with command bit names.
   // All OCmds/MCmds and ORdys/MRdys are now Local Tags.
   // Added Sts_RdyAck and Sts_RdyReset for use by containing objects.
   // Modified to remove Suppressed from the conditions which show
   // the "Inhibited" breadcrumb.
   // Added Inp_OoS for Out of Service from parent object's P_CmdSrc.
   // V4.10.00  2019-03-08:  Unmodified, up-rev only for Library 4.10.00
   // ============================================================
   // This instruction monitors one input condition and provides one Alarm with:
   //   * configurable latching (reset required) and acknowledgement requirement
   //   * configurable alarm severity
   // 1..250 = Low  (blue, typ. informational)
   // 251-500 = Medium  (yelllow, typ. warning)
   // 501-750 = High  (red, typ. process exception)
   // 751-1000 = Urgent  (magenta, typ. equip. fault)
   // * configurable minimum ON time (e.g., to ensure it is seen by the HMI)
   // * commands to suppress/unsuppress (Prog), shelve/unshelve (Oper)
   // and disable/enable (Maint) the alarm.
   // * configurable amount of time shelved to automatically unshelve an alarm
   // * FTA&E support for suppressed, shelved and disabled states (V7.0)
   // NOTE regarding parameter naming:
   // FTA&E names (same as ALMD instruction) are used instead
   // of the ANSI/ISA 18.2-2016 names, as follows:
   // "Disabled" is the equivalent of "Out of Service" in ISA 18.2.
   // (the Disabled state is owned by Maintenance)
   // "Suppressed" is the equivalent of "Suppressed by Design" in ISA 18.2.
   // (the Suppressed state is owned by Program logic)
   // "Shelved" is the same as in ISA 18.2.
   // (the Shelved state is owned by Operator, but may be cleared
   // by Program logic based on time, shift change, etc.)
   // This instruction is usually nested within other instructions, with one instance
   // used for each Alarm generated by the containing instruction.  It may also be
   // used as a standalone instruction for Alarm conditions generated by custom logic.
   // ________________________________________
   // FTAE Alarm Setup:
   // ________________________________________
   // (object).(alarm).Com_AE.0:  Alarm to FTAE
   // .Com_AE.1:   Ack to/from FTAE
   // .Com_AE.2:  Out of Service (from object's P_CmdSrc)
   // .Com_AE.3:   Shelved from FTAE Status
   // .Com_AE.4:   Shelve/Reshelve to FTAE Control (auto reset)
   // .Com_AE.5:   Unshelve to FTAE Control (auto reset)
   // .Com_AE.6:   Suppressed from FTAE Status
   // .Com_AE.7:   Suppress to FTAE Control (auto reset)
   // .Com_AE.8:   Unsuppress to FTAE Control (auto reset)
   // .Com_AE.9:   Disabled from FTAE Status
   // .Com_AE.10: Disable to FTAE Control (auto reset)
   // .Com_AE.11: Enable to FTAE Control (auto reset)
   // all other bits unused
   //     .Cfg_MaxShelfT is also used in FTAE config.
   // .Cfg_Severity is used by FTAE in FTView 8.x.
   // ============================================================
   // POWERUP / INVALID STATE HANDLING
   // ============================================================
   // All internal Work (state) bits maintain states through a power cycle and are
   // independent.  No first-scan logic is required.  See the Prescan routine for
   // powerup / prescan code.
   // ============================================================
   // SHOW LOCAL STRINGS
   // ============================================================
   // The STRINGs containing the text associated with each instance of this
   // instruction cannot be Input or Output Parameters, because STRINGs are not
   //  'atomic' types. (Inputs and Outputs must be SINT, INT, DINT, REAL, or BOOL.)
   // In order to make it easier to find and configure these STRINGs, this rung
   // was added.  THE JMP (and the LBL on the following rung)
   // MUST NOT BE REMOVED!!!
   // To view the STRINGs, go to the instruction instance (in LD or FBD), RIGHT-click
   // to bring up the context menu and select "Open Instruction Logic".
   // This rung will appear with the STRING values for the selected instance.
   // You may double-click the STRING values here to modify them as well.
   0: JMP(SkipText)LOWER(Cfg_Tag,Cfg_Cond)LOWER(HMI_Lib,HMI_Type);
   // ============================================================
   // CONFIGURATION
   // ============================================================
   // In the object containing this alarm, other configuration (such as not having
   // any limit switches) may make this particular alarm meaningless.
   // The Program Configuration "Allow Exist" is used to hide this alarm
   // on the object's faceplate and other graphics, and forces the Cfg_Exist to 0.
   1: LBL(SkipText)XIO(PCfg_AllowExist)OTU(Cfg_Exists);
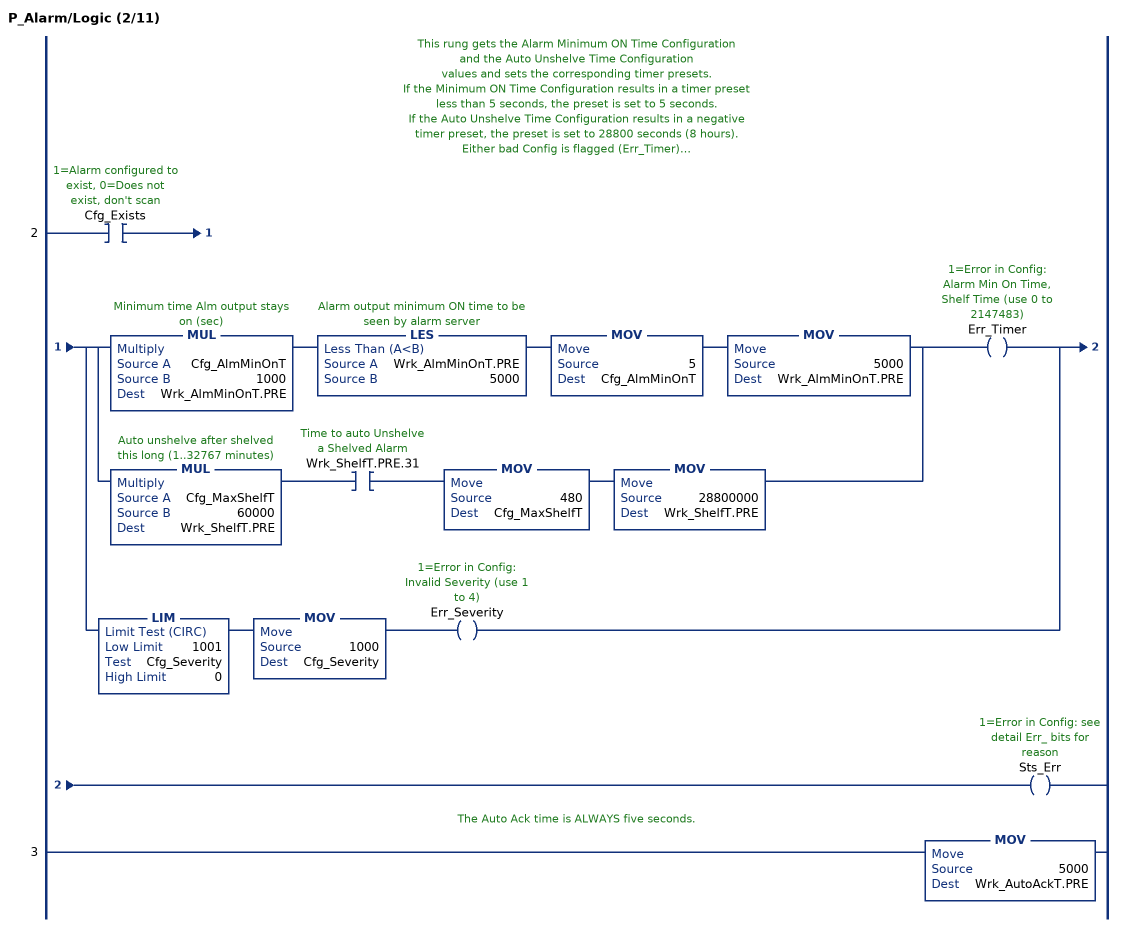
   // This rung gets the Alarm Minimum ON Time Configuration
   // and the Auto Unshelve Time Configuration
   // values and sets the corresponding timer presets.
   // If the Minimum ON Time Configuration results in a timer preset
   // less than 5 seconds, the preset is set to 5 seconds.
   // If the Auto Unshelve Time Configuration results in a negative
   // timer preset, the preset is set to 28800 seconds (8 hours).
   // Either bad Config is flagged (Err_Timer).
   // Bad Config is also flagged if the Cfg_Severity is out of range (valid = 1..1000) (Err_Severity).
   2: XIC(Cfg_Exists)[[MUL(Cfg_AlmMinOnT,1000,Wrk_AlmMinOnT.PRE) LES(Wrk_AlmMinOnT.PRE,5000) MOV(5,Cfg_AlmMinOnT) MOV(5000,Wrk_AlmMinOnT.PRE) ,MUL(Cfg_MaxShelfT,60000,Wrk_ShelfT.PRE) XIC(Wrk_ShelfT.PRE.31) MOV(480,Cfg_MaxShelfT) MOV(28800000,Wrk_ShelfT.PRE) ] OTE(Err_Timer) ,LIM(1001,Cfg_Severity,0) MOV(1000,Cfg_Severity) OTE(Err_Severity) ]OTE(Sts_Err);
   // The Auto Ack time is ALWAYS five seconds.
   3: MOV(5000,Wrk_AutoAckT.PRE);
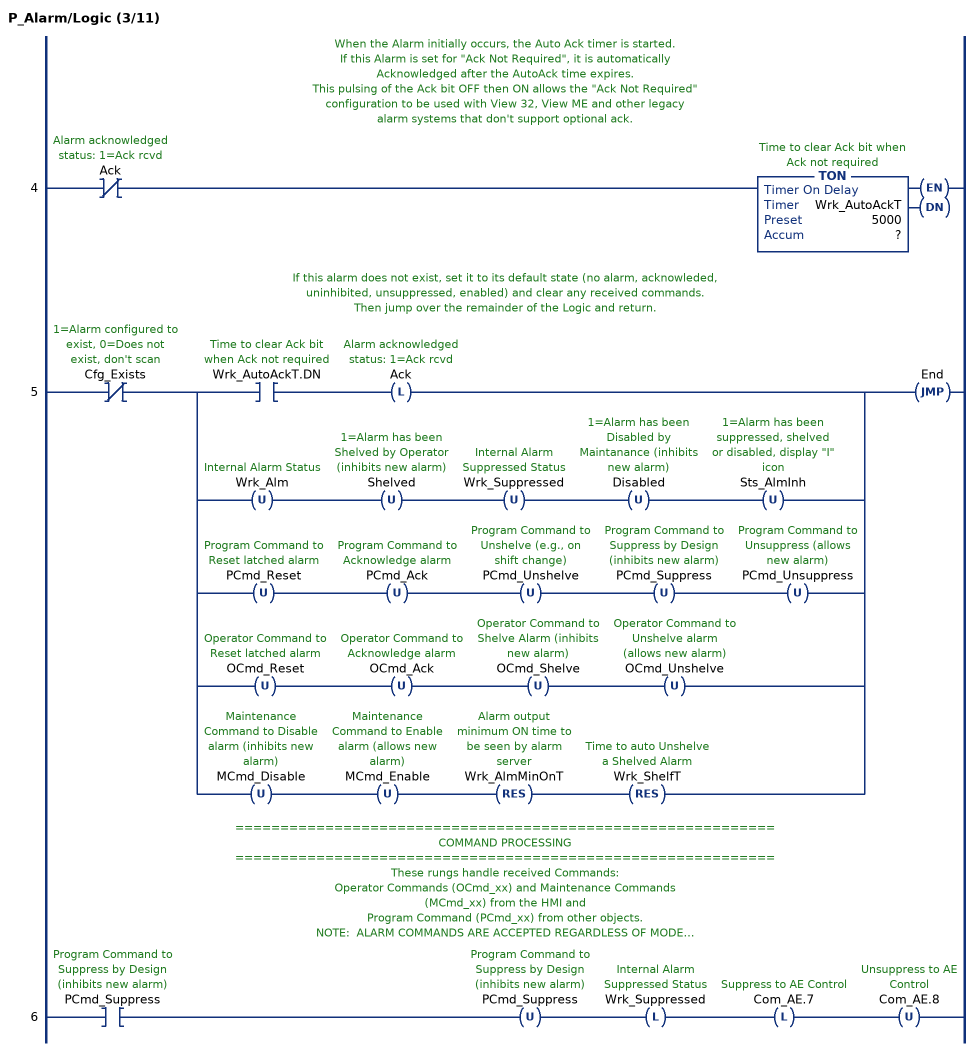
   // When the Alarm initially occurs, the Auto Ack timer is started.
   // If this Alarm is set for "Ack Not Required", it is automatically
   // Acknowledged after the AutoAck time expires.
   // This pulsing of the Ack bit OFF then ON allows the "Ack Not Required"
   // configuration to be used with View 32, View ME and other legacy
   // alarm systems that don't support optional ack.
   4: XIO(Ack)TON(Wrk_AutoAckT,?,?);
   // If this alarm does not exist, set it to its default state (no alarm, acknowleded,
   // uninhibited, unsuppressed, enabled) and clear any received commands.
   // Then jump over the remainder of the Logic and return.
   5: XIO(Cfg_Exists)[XIC(Wrk_AutoAckT.DN) OTL(Ack) ,OTU(Wrk_Alm) OTU(Shelved) OTU(Wrk_Suppressed) OTU(Disabled) OTU(Sts_AlmInh) ,OTU(PCmd_Reset) OTU(PCmd_Ack) OTU(PCmd_Unshelve) OTU(PCmd_Suppress) OTU(PCmd_Unsuppress) ,OTU(OCmd_Reset) OTU(OCmd_Ack) OTU(OCmd_Shelve) OTU(OCmd_Unshelve) ,OTU(MCmd_Disable) OTU(MCmd_Enable) RES(Wrk_AlmMinOnT) RES(Wrk_ShelfT) ]JMP(End);
   // ============================================================
   // COMMAND PROCESSING
   // ============================================================
   // These rungs handle received Commands:
   // Operator Commands (OCmd_xx) and Maintenance Commands
   // (MCmd_xx) from the HMI and
   // Program Command (PCmd_xx) from other objects.
   // NOTE:  ALARM COMMANDS ARE ACCEPTED REGARDLESS OF MODE.
   // This rung receives the Program Alarm Inhibit Command.
   // If configured for EDGE, the Command is cleared.
   // #####  V4.00.00  2018-06-07:  Deleted Cfg_PCmdClear; all Program Commands are now self-clearing.  #####
   6: XIC(PCmd_Suppress)OTU(PCmd_Suppress)OTL(Wrk_Suppressed)OTL(Com_AE.7)OTU(Com_AE.8);
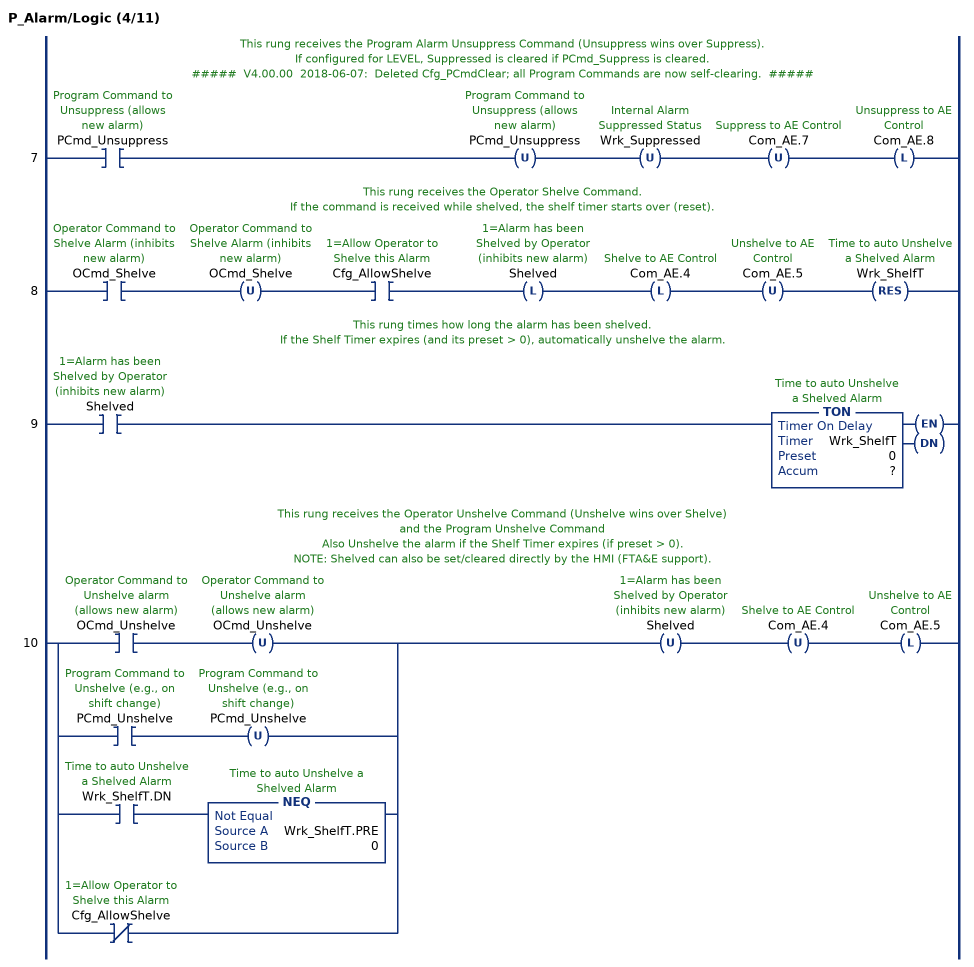
   // This rung receives the Program Alarm Unsuppress Command (Unsuppress wins over Suppress).
   // If configured for LEVEL, Suppressed is cleared if PCmd_Suppress is cleared.
   // #####  V4.00.00  2018-06-07:  Deleted Cfg_PCmdClear; all Program Commands are now self-clearing.  #####
   7: XIC(PCmd_Unsuppress)OTU(PCmd_Unsuppress)OTU(Wrk_Suppressed)OTU(Com_AE.7)OTL(Com_AE.8);
   // This rung receives the Operator Shelve Command.
   // If the command is received while shelved, the shelf timer starts over (reset).
   8: XIC(OCmd_Shelve)OTU(OCmd_Shelve)XIC(Cfg_AllowShelve)OTL(Shelved)OTL(Com_AE.4)OTU(Com_AE.5)RES(Wrk_ShelfT);
   // This rung times how long the alarm has been shelved.
   // If the Shelf Timer expires (and its preset > 0), automatically unshelve the alarm.
   9: XIC(Shelved)TON(Wrk_ShelfT,?,?);
   // This rung receives the Operator Unshelve Command (Unshelve wins over Shelve)
   // and the Program Unshelve Command
   // Also Unshelve the alarm if the Shelf Timer expires (if preset > 0).
   // NOTE: Shelved can also be set/cleared directly by the HMI (FTA&E support).
   10: [XIC(OCmd_Unshelve) OTU(OCmd_Unshelve) ,XIC(PCmd_Unshelve) OTU(PCmd_Unshelve) ,XIC(Wrk_ShelfT.DN) NEQ(Wrk_ShelfT.PRE,0) ,XIO(Cfg_AllowShelve) ]OTU(Shelved)OTU(Com_AE.4)OTL(Com_AE.5);
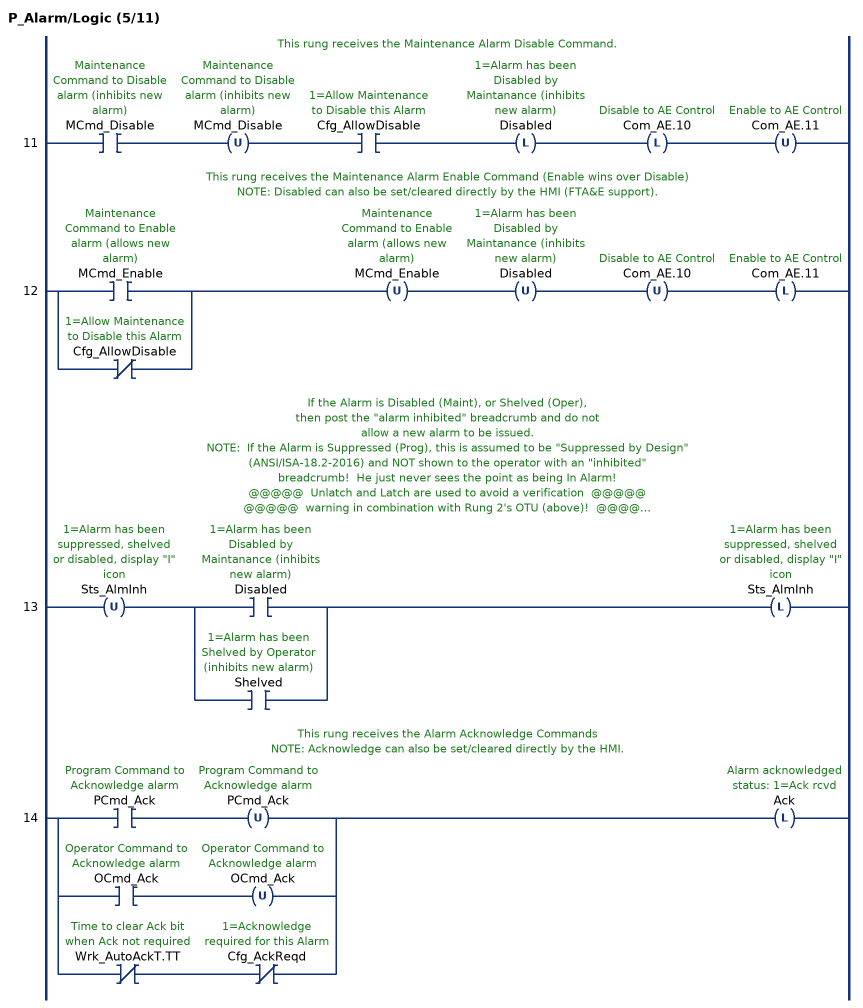
   // This rung receives the Maintenance Alarm Disable Command.
   11: XIC(MCmd_Disable)OTU(MCmd_Disable)XIC(Cfg_AllowDisable)OTL(Disabled)OTL(Com_AE.10)OTU(Com_AE.11);
   // This rung receives the Maintenance Alarm Enable Command (Enable wins over Disable)
   // NOTE: Disabled can also be set/cleared directly by the HMI (FTA&E support).
   12: [XIC(MCmd_Enable) ,XIO(Cfg_AllowDisable) ]OTU(MCmd_Enable)OTU(Disabled)OTU(Com_AE.10)OTL(Com_AE.11);
   // If the Alarm is Disabled (Maint), or Shelved (Oper),
   // then post the "alarm inhibited" breadcrumb and do not
   // allow a new alarm to be issued.
   // NOTE:  If the Alarm is Suppressed (Prog), this is assumed to be "Suppressed by Design"
   // (ANSI/ISA-18.2-2016) and NOT shown to the operator with an "inhibited"
   // breadcrumb!  He just never sees the point as being In Alarm!
   // @@@@@  Unlatch and Latch are used to avoid a verification  @@@@@
   // @@@@@  warning in combination with Rung 2's OTU (above)!  @@@@@
   // #####  V4.00.00  2018-06-07:  Modified to remove Suppressed from the conditions to show the "Inhibited" breadcrumb.  #####
   13: OTU(Sts_AlmInh)[XIC(Disabled) ,XIC(Shelved) ]OTL(Sts_AlmInh);
   // This rung receives the Alarm Acknowledge Commands
   // NOTE: Acknowledge can also be set/cleared directly by the HMI.
   14: [XIC(PCmd_Ack) OTU(PCmd_Ack) ,XIC(OCmd_Ack) OTU(OCmd_Ack) ,XIO(Wrk_AutoAckT.TT) XIO(Cfg_AckReqd) ]OTL(Ack);
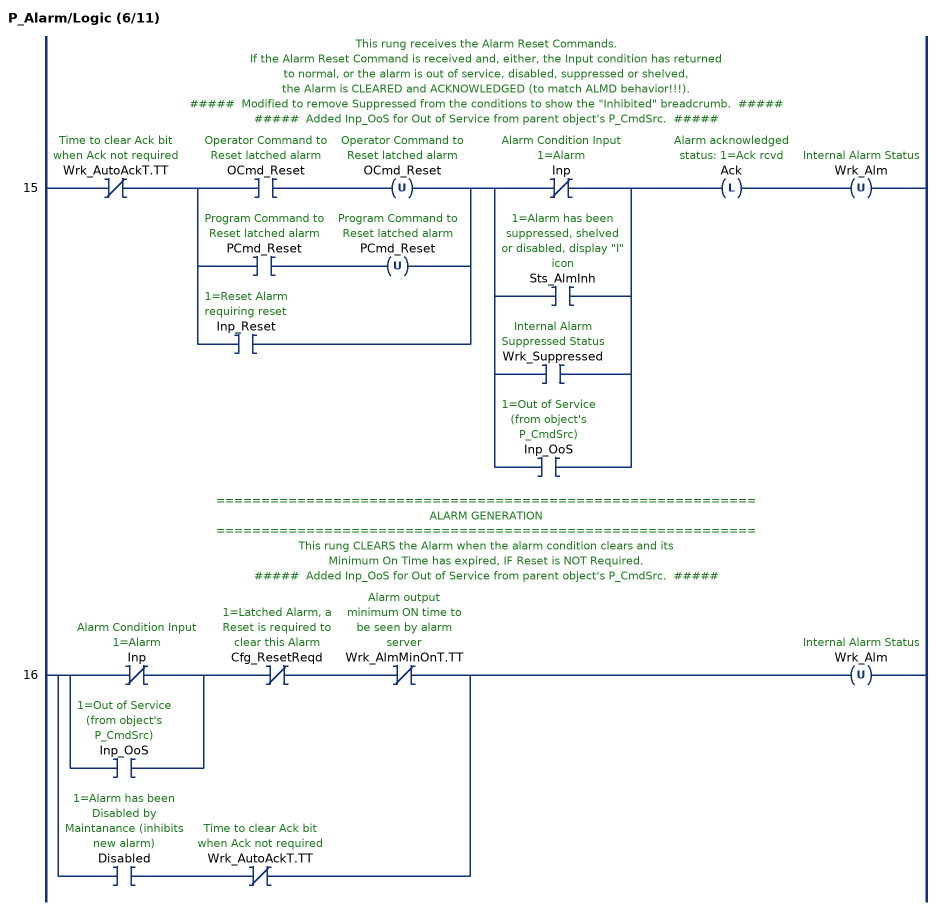
   // This rung receives the Alarm Reset Commands.
   // If the Alarm Reset Command is received and, either, the Input condition has returned
   // to normal, or the alarm is out of service, disabled, suppressed or shelved,
   // the Alarm is CLEARED and ACKNOWLEDGED (to match ALMD behavior!!!).
   // #####  Modified to remove Suppressed from the conditions to show the "Inhibited" breadcrumb.  #####
   // #####  Added Inp_OoS for Out of Service from parent object's P_CmdSrc.  #####
   15: XIO(Wrk_AutoAckT.TT)[XIC(OCmd_Reset) OTU(OCmd_Reset) ,XIC(PCmd_Reset) OTU(PCmd_Reset) ,XIC(Inp_Reset) ][XIO(Inp) ,XIC(Sts_AlmInh) ,XIC(Wrk_Suppressed) ,XIC(Inp_OoS) ]OTL(Ack)OTU(Wrk_Alm);
   // ============================================================
   // ALARM GENERATION
   // ============================================================
   // This rung CLEARS the Alarm when the alarm condition clears and its
   // Minimum On Time has expired, IF Reset is NOT Required.
   // #####  Added Inp_OoS for Out of Service from parent object's P_CmdSrc.  #####
   16: [[XIO(Inp) ,XIC(Inp_OoS) ] XIO(Cfg_ResetReqd) XIO(Wrk_AlmMinOnT.TT) ,XIC(Disabled) XIO(Wrk_AutoAckT.TT) ]OTU(Wrk_Alm);
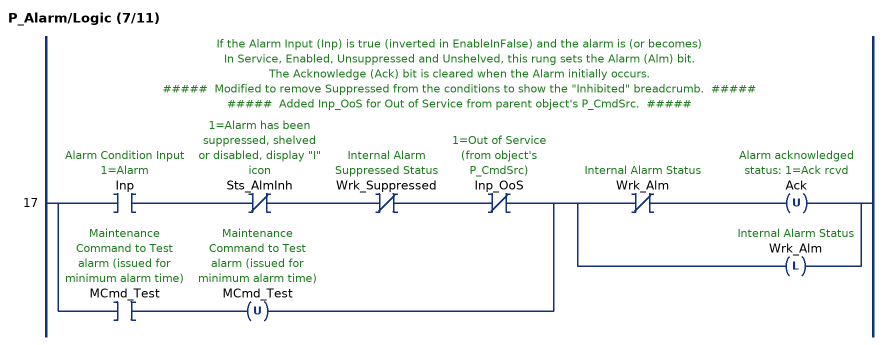
   // If the Alarm Input (Inp) is true (inverted in EnableInFalse) and the alarm is (or becomes)
   // In Service, Enabled, Unsuppressed and Unshelved, this rung sets the Alarm (Alm) bit.
   // The Acknowledge (Ack) bit is cleared when the Alarm initially occurs.
   // #####  Modified to remove Suppressed from the conditions to show the "Inhibited" breadcrumb.  #####
   // #####  Added Inp_OoS for Out of Service from parent object's P_CmdSrc.  #####
   17: [XIC(Inp) XIO(Sts_AlmInh) XIO(Wrk_Suppressed) XIO(Inp_OoS) ,XIC(MCmd_Test) OTU(MCmd_Test) ][XIO(Wrk_Alm) OTU(Ack) ,OTL(Wrk_Alm) ];
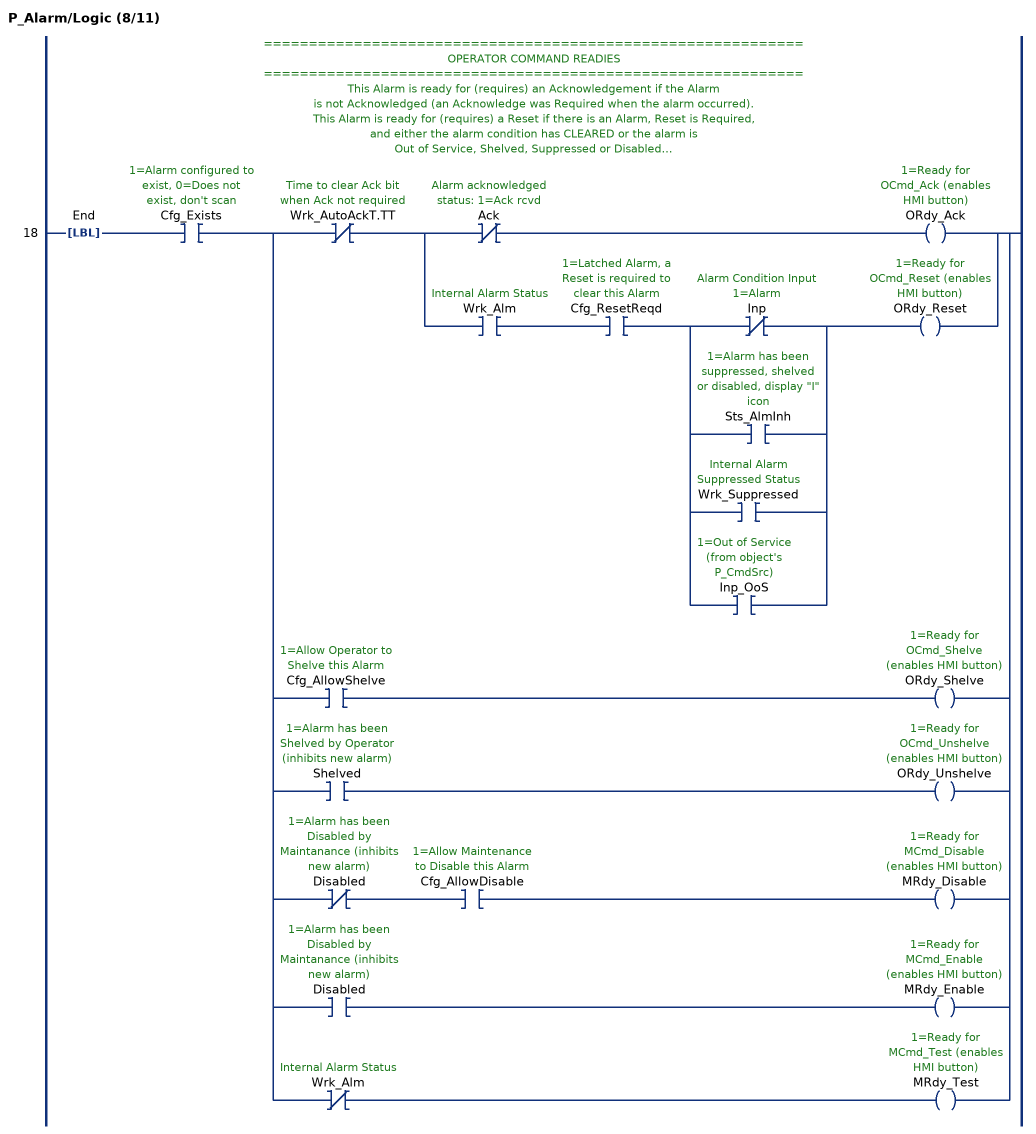
   // ============================================================
   // OPERATOR COMMAND READIES
   // ============================================================
   // This Alarm is ready for (requires) an Acknowledgement if the Alarm
   // is not Acknowledged (an Acknowledge was Required when the alarm occurred).
   // This Alarm is ready for (requires) a Reset if there is an Alarm, Reset is Required,
   // and either the alarm condition has CLEARED or the alarm is
   // Out of Service, Shelved, Suppressed or Disabled.
   // .
   // If the Alarm is NOT Shelved, it is ready for Shelve.
   // If the Alarm IS Shelved, it is ready for Unshelve.
   // If the Alarm is NOT Disabled, it is ready for Disable.
   // If the Alarm IS Disabled, it is ready for Enable.
   // NOTE: This rung appears before the Values/Status rung because the Rdy_Reset
   // condition is used to eliminate redundant logic in the rung below for Val_Notify.0.
   // #####  V4.00.00  2018-06-07:  Aligned ready bit naming with command bit names.  #####
   // #####  All OCmds/MCmds and ORdys/MRdys are now Local Tags.  #####
   // #####  Added Sts_RdyAck and Sts_ResetReqd for use by containing objects.  #####
   // #####  Modified to remove Suppressed from the conditions to show the "Inhibited" breadcrumb.  #####
   // #####  Added Inp_OoS for Out of Service from parent object's P_CmdSrc.  #####
   18: LBL(End)XIC(Cfg_Exists)[XIO(Wrk_AutoAckT.TT) [XIO(Ack) OTE(ORdy_Ack) ,XIC(Wrk_Alm) XIC(Cfg_ResetReqd) [XIO(Inp) ,XIC(Sts_AlmInh) ,XIC(Wrk_Suppressed) ,XIC(Inp_OoS) ] OTE(ORdy_Reset) ] ,XIC(Cfg_AllowShelve) OTE(ORdy_Shelve) ,XIC(Shelved) OTE(ORdy_Unshelve) ,XIO(Disabled) XIC(Cfg_AllowDisable) OTE(MRdy_Disable) ,XIC(Disabled) OTE(MRdy_Enable) ,XIO(Wrk_Alm) OTE(MRdy_Test) ];
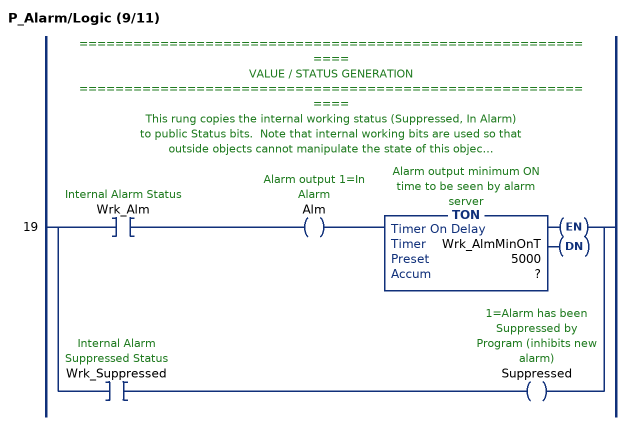
   // ============================================================
   // VALUE / STATUS GENERATION
   // ============================================================
   // This rung copies the internal working status (Suppressed, In Alarm)
   // to public Status bits.  Note that internal working bits are used so that
   // outside objects cannot manipulate the state of this object
   // by setting/clearing its Status and Alarm bits.
   // Public Status is generated for:
   // Alarm (with minimum ON time to be seen by polling)
   // Alarm Suppressed
   // Unsuppressed, Unshelved and Enabled are generated for HMI (FTVSE 7).
   // (Ack, Shelved and Disabled can be set/cleared by the HMI directly.
   // Note that these bits are "read/write" outputs in the parameter definition.)
   19: [XIC(Wrk_Alm) OTE(Alm) TON(Wrk_AlmMinOnT,?,?) ,XIC(Wrk_Suppressed) OTE(Suppressed) ];
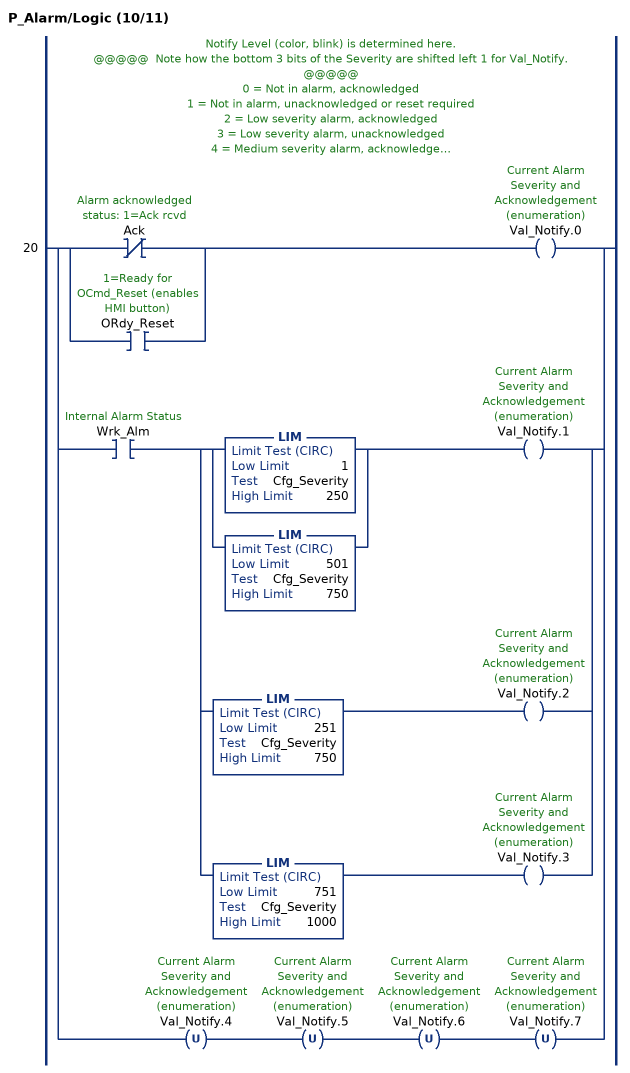
   // Notify Level (color, blink) is determined here.
   // @@@@@  Note how the bottom 3 bits of the Severity are shifted left 1 for Val_Notify.  @@@@@
   // 0 = Not in alarm, acknowledged
   // 1 = Not in alarm, unacknowledged or reset required
   // 2 = Low severity alarm, acknowledged
   // 3 = Low severity alarm, unacknowledged
   // 4 = Medium severity alarm, acknowledged
   // 5 = Medium severity alarm, unacknowledged
   // 6 = High severity alarm, acknowledged
   // 7 = High severity alarm, unacknowledged
   // 8 = Urgent severity alarm, acknowledged
   // 9 = Urgent severity alarm, unacknowledged
   // NOTE that the alarm bell icon will blink, even though the alarm is Acknowledged,
   // if an Alarm Reset is required (to get the Operator's attention).
   20: [[XIO(Ack) ,XIC(ORdy_Reset) ] OTE(Val_Notify.0) ,XIC(Wrk_Alm) [[LIM(1,Cfg_Severity,250) ,LIM(501,Cfg_Severity,750) ] OTE(Val_Notify.1) ,LIM(251,Cfg_Severity,750) OTE(Val_Notify.2) ,LIM(751,Cfg_Severity,1000) OTE(Val_Notify.3) ] ,OTU(Val_Notify.4) OTU(Val_Notify.5) OTU(Val_Notify.6) OTU(Val_Notify.7) ];
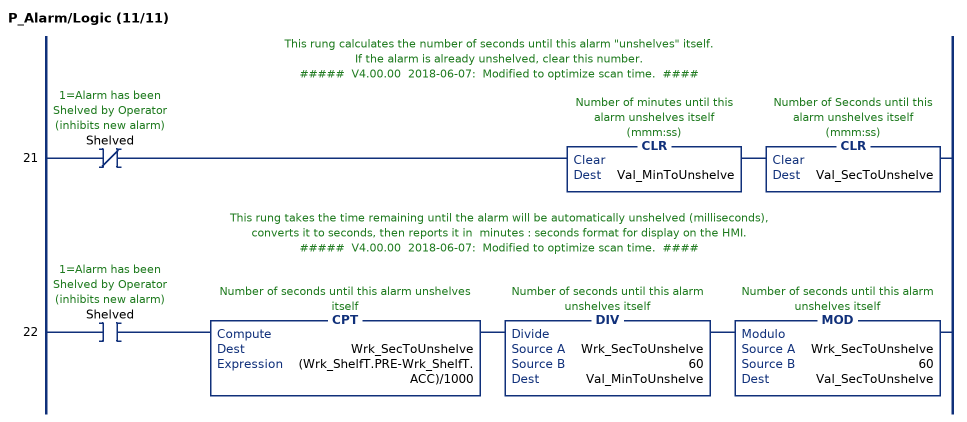
   // This rung calculates the number of seconds until this alarm "unshelves" itself.
   // If the alarm is already unshelved, clear this number.
   // #####  V4.00.00  2018-06-07:  Modified to optimize scan time.  ####
   21: XIO(Shelved)CLR(Val_MinToUnshelve)CLR(Val_SecToUnshelve);
   // This rung takes the time remaining until the alarm will be automatically unshelved (milliseconds),
   // converts it to seconds, then reports it in  minutes : seconds format for display on the HMI.
   // #####  V4.00.00  2018-06-07:  Modified to optimize scan time.  ####
   22: XIC(Shelved)CPT(Wrk_SecToUnshelve,(Wrk_ShelfT.PRE-Wrk_ShelfT.ACC)/1000)DIV(Wrk_SecToUnshelve,60,Val_MinToUnshelve)MOD(Wrk_SecToUnshelve,60,Val_SecToUnshelve);
END_ROUTINE
